// TIA Portal V16 export
// export: Created 2023-03-29T11:04:42.9092008Z, ExportSetting WithDefaults, DisplayName Totally Integrated Automation Portal, DisplayVersion V16 Update 6, DisplayName TIA Portal Version Control Interface, DisplayVersion V16 Update 2, DisplayName TIA Portal Openness, DisplayVersion V16 Update 6, DisplayName STEP 7 Professional, DisplayVersion V16 Update 6, DisplayName STEP 7 Safety, DisplayVersion V16, DisplayName WinCC Advanced, DisplayVersion V16 Update 6
FUNCTION "Convert_analogs" : Void   // FC14, LAD
TITLE = Funkcja konwertera analogów
{ S7_Optimized_Access := 'TRUE' }
AUTHOR : RTecmer
VERSION : 0.1
// "Switch_set_OverCurrentInverer" - Porzełączni wyboru źródła wartości parametrówą falownika  ( 0- wartość z Modbus RTU, 1- wartość zadana ręcznie) / Konwertowanie zmiennych procesowych
// stored: AutoNumber true, IsIECCheckEnabled false, SetENOAutomatically false, UDAEnableTagReadback false
   VAR_TEMP   // added for the SCL form of the ladder/FBD networks
      _w1 : Bool;
   END_VAR
BEGIN

REGION Network 1: Przepywomierz Q1 Pompownia
   // Pobrane z Modbus RTU
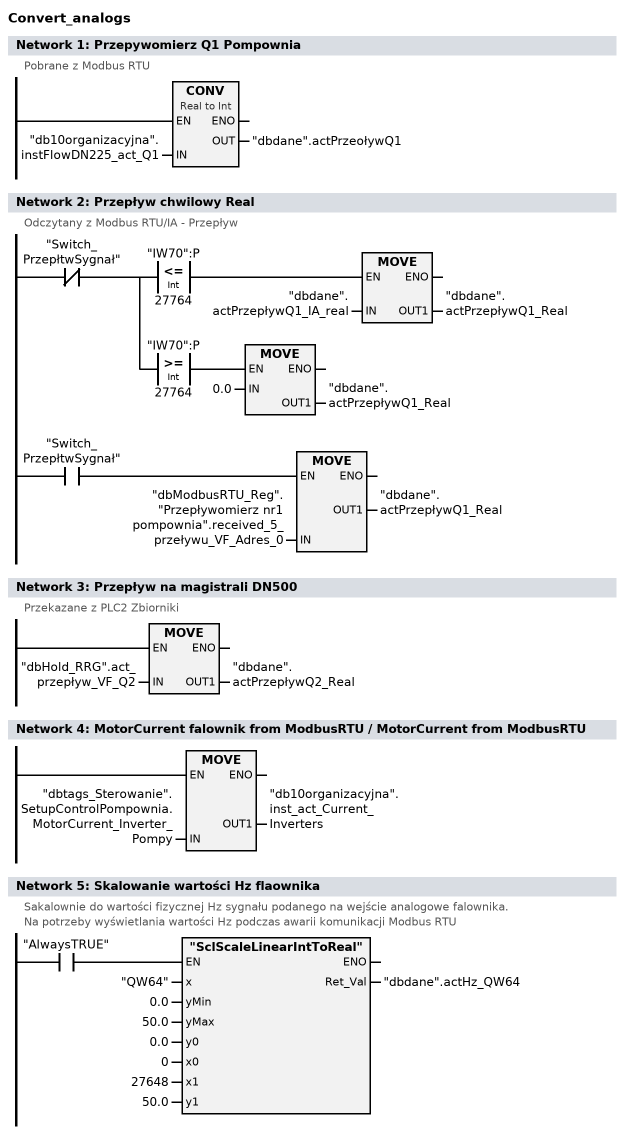
   RUNG wire#powerrail
      { S7_Templates := "[SrcType := Real, DestType := Int]" } Convert(in := "db10organizacyjna".instFlowDN225_act_Q1, out => "dbdane".actPrzeoływQ1)
   END_RUNG
   // the same network as SCL:
   "dbdane".actPrzeoływQ1 := REAL_TO_INT("db10organizacyjna".instFlowDN225_act_Q1);
END_REGION

REGION Network 2: Przepływ chwilowy Real
   // Odczytany z Modbus RTU/IA - Przepływ
   RUNG wire#powerrail
      I_Contact( "Switch_PrzepłtwSygnał" )
      wire#w1
      { S7_Templates := "SrcType := Int" } LE_Contact(in1 := "IW70":P, in2 := 27764)
      Move(in := "dbdane".actPrzepływQ1_IA_real, out1 => "dbdane".actPrzepływQ1_Real)
   END_RUNG
   RUNG wire#w1
      { S7_Templates := "SrcType := Int" } GE_Contact(in1 := "IW70":P, in2 := 27764)
      Move(in := 0.0, out1 => "dbdane".actPrzepływQ1_Real)
   END_RUNG
   RUNG wire#powerrail
      Contact( "Switch_PrzepłtwSygnał" )
      Move(in := "dbModbusRTU_Reg"."Przepływomierz nr1 pompownia".received_5_przeływu_VF_Adres_0, out1 => "dbdane".actPrzepływQ1_Real)
   END_RUNG
   // the same network as SCL:
   #_w1 := NOT "Switch_PrzepłtwSygnał";
   IF #_w1 AND ("IW70":P <= 27764) THEN
       "dbdane".actPrzepływQ1_Real := "dbdane".actPrzepływQ1_IA_real;
   END_IF;
   IF #_w1 AND ("IW70":P >= 27764) THEN "dbdane".actPrzepływQ1_Real := 0.0; END_IF;
   IF "Switch_PrzepłtwSygnał" THEN
       "dbdane".actPrzepływQ1_Real := "dbModbusRTU_Reg"."Przepływomierz nr1 pompownia".received_5_przeływu_VF_Adres_0;
   END_IF;
END_REGION

REGION Network 3: Przepływ na magistrali DN500
   // Przekazane z PLC2 Zbiorniki
   RUNG wire#powerrail
      Move(in := "dbHold_RRG".act_przepływ_VF_Q2, out1 => "dbdane".actPrzepływQ2_Real)
   END_RUNG
   // the same network as SCL:
   "dbdane".actPrzepływQ2_Real := "dbHold_RRG".act_przepływ_VF_Q2;
END_REGION

REGION Network 4: MotorCurrent falownik from ModbusRTU / MotorCurrent from ModbusRTU
   RUNG wire#powerrail
      Move(in := "dbtags_Sterowanie".SetupControlPompownia.MotorCurrent_Inverter_Pompy, out1 => "db10organizacyjna".inst_act_Current_Inverters)
   END_RUNG
   // the same network as SCL:
   "db10organizacyjna".inst_act_Current_Inverters := "dbtags_Sterowanie".SetupControlPompownia.MotorCurrent_Inverter_Pompy;
END_REGION

REGION Network 5: Skalowanie wartości Hz flaownika
   // Sakalownie do wartości fizycznej Hz sygnału podanego na wejście analogowe falownika.
   // Na potrzeby wyświetlania wartości Hz podczas awarii komunikacji Modbus RTU
   RUNG wire#powerrail
      Contact( "AlwaysTRUE" )
      "SclScaleLinearIntToReal"(x := "QW64", yMin := 0.0, yMax := 50.0, y0 := 0.0, x0 := 0, x1 := 27648, y1 := 50.0, Ret_Val => "dbdane".actHz_QW64)
   END_RUNG
   // the same network as SCL:
   IF "AlwaysTRUE" THEN
       "dbdane".actHz_QW64 := "SclScaleLinearIntToReal"(x := "QW64",
                               yMin := 0.0,
                               yMax := 50.0,
                               y0 := 0.0,
                               x0 := 0,
                               x1 := 27648,
                               y1 := 50.0);
   END_IF;
END_REGION
END_FUNCTION
